FUNCTION_BLOCK FB_System_WP_946
VAR_INPUT
	Freigabe_auto			: BOOL;
	Freigabe_Deakt_auto 	: BOOL;
	Betrieb_Anford_auto		: BOOL;
END_VAR
VAR_OUTPUT
	{attribute 'OPC.UA.DA' := '1'}Steuerung				: ST_System_WP_Steuerung;	
	{attribute 'OPC.UA.DA' := '1'}Stellwert				: ST_System_WP_Stellwert;	
	{attribute 'OPC.UA.DA' := '1'}Zustand					: ST_System_WP_Zustand;	
	{attribute 'OPC.UA.DA' := '1'}Parameter				: ST_System_WP_Parameter;	
END_VAR
VAR
	Waermepumpe_946			: FB_WP;
	Zustandscheck			: FB_System_WP_Zustandscheck;
	Logik					: FB_System_WP_Logik;
	Ablaufsteuerung			: FB_System_WP_Ablaufsteuerung;

	SV_146: FB_SV;
	SV_246: FB_SV;
END_VAR
VAR // added by the converter: edge detectors and wires of the graphical bodies
    _w1, _w2, _w3, _w4 : ANY;
END_VAR

// note: this text did not pass the execution check against the stored diagram
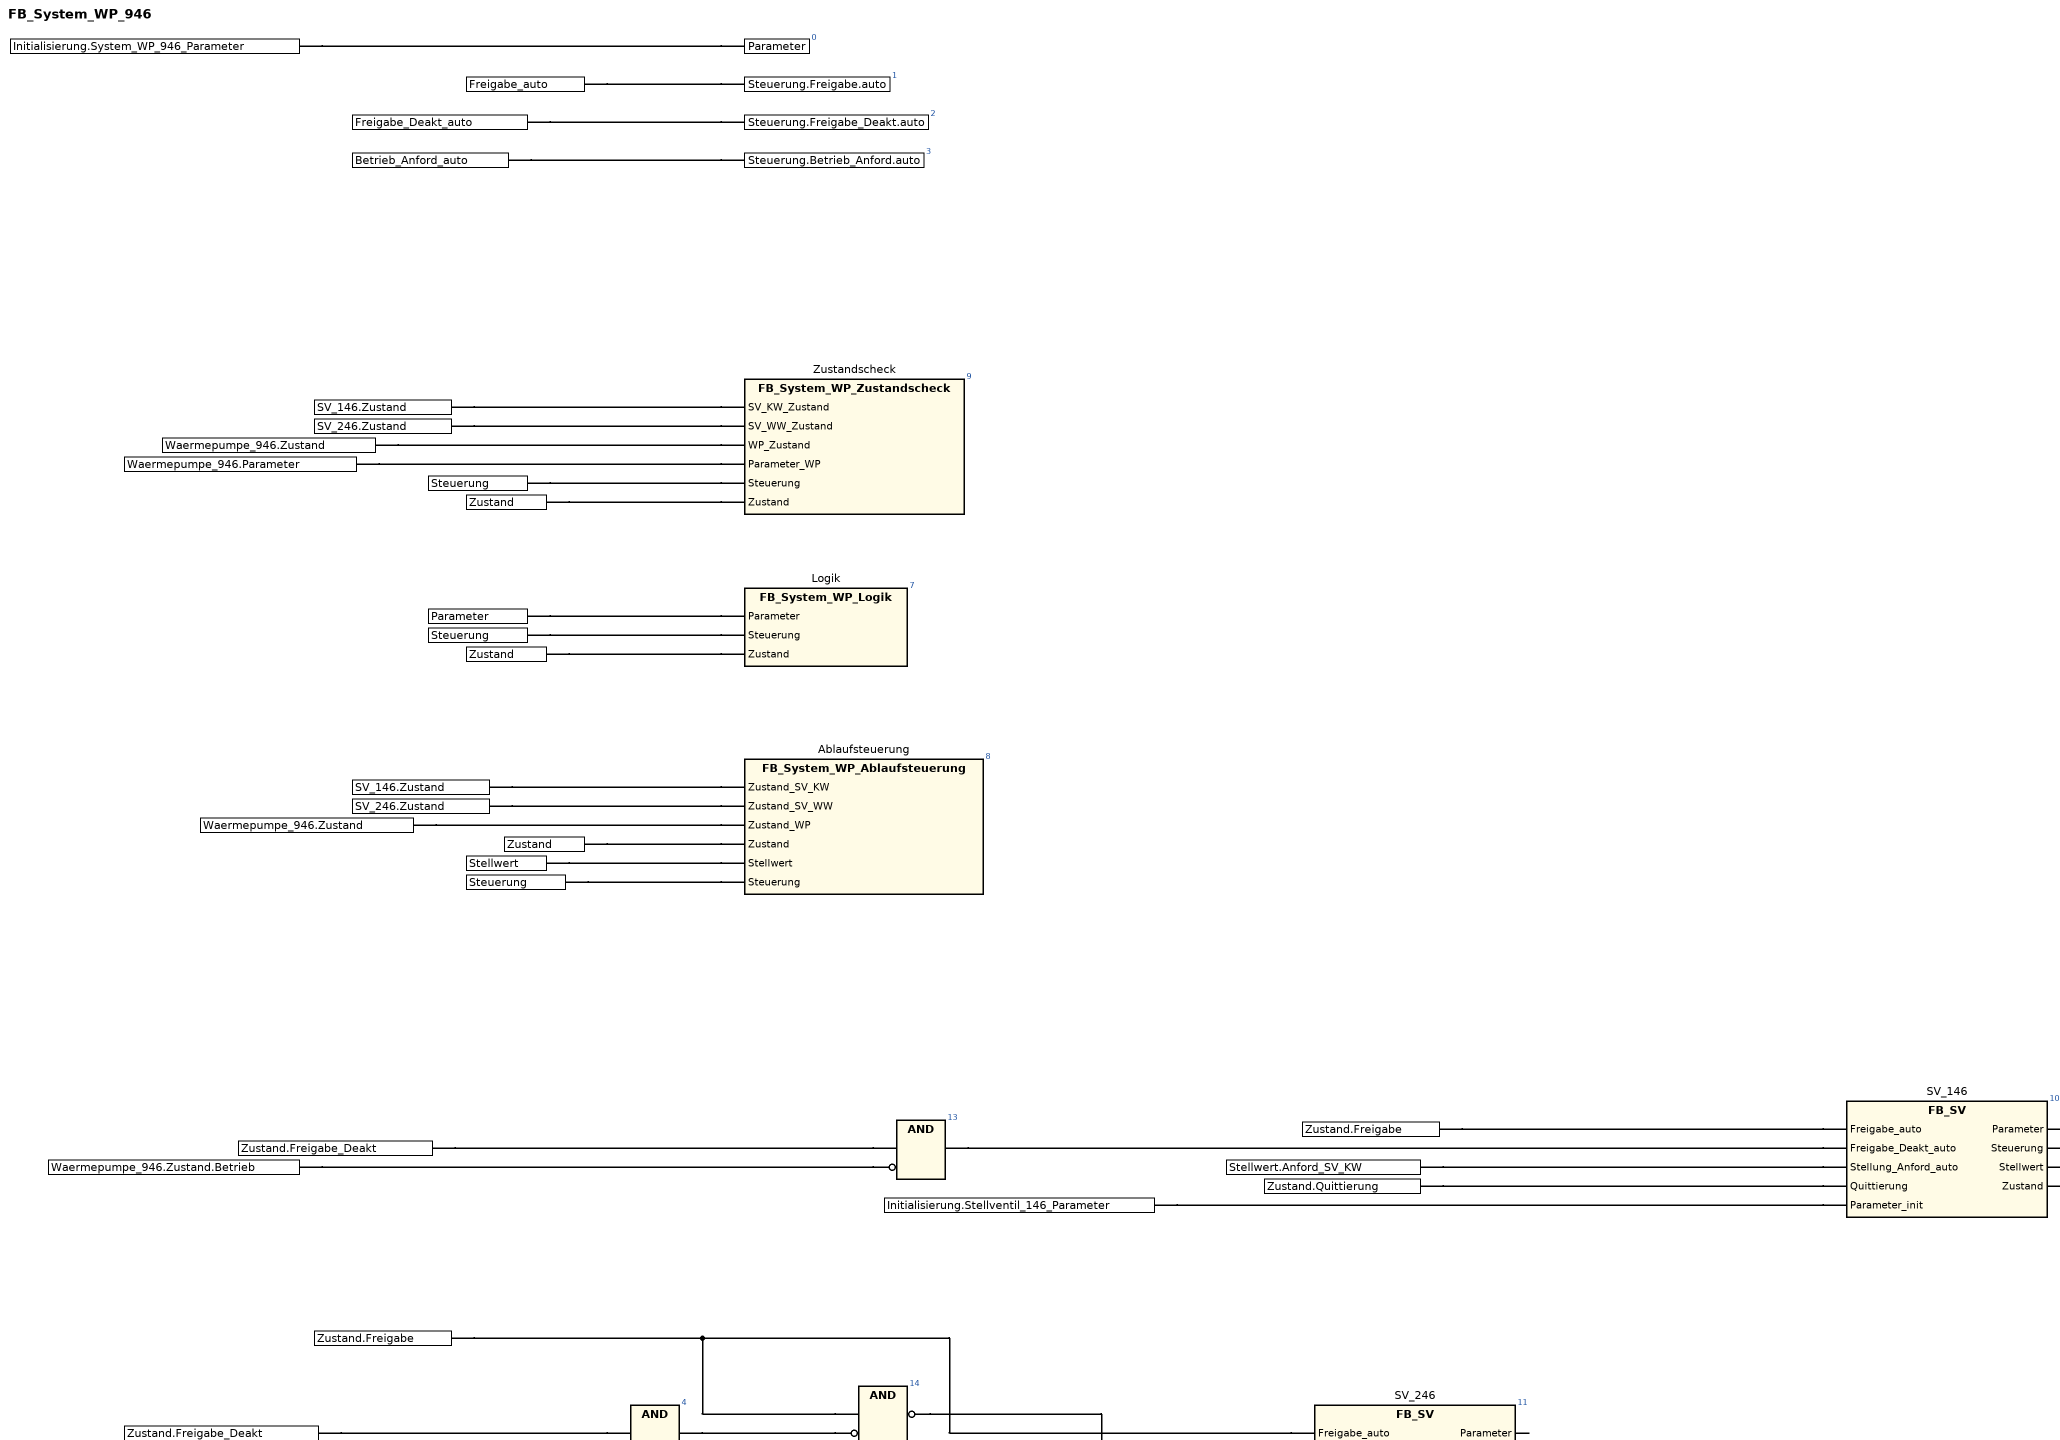
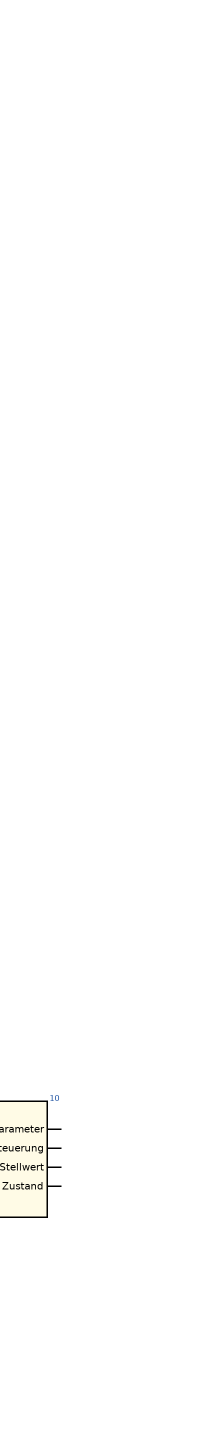
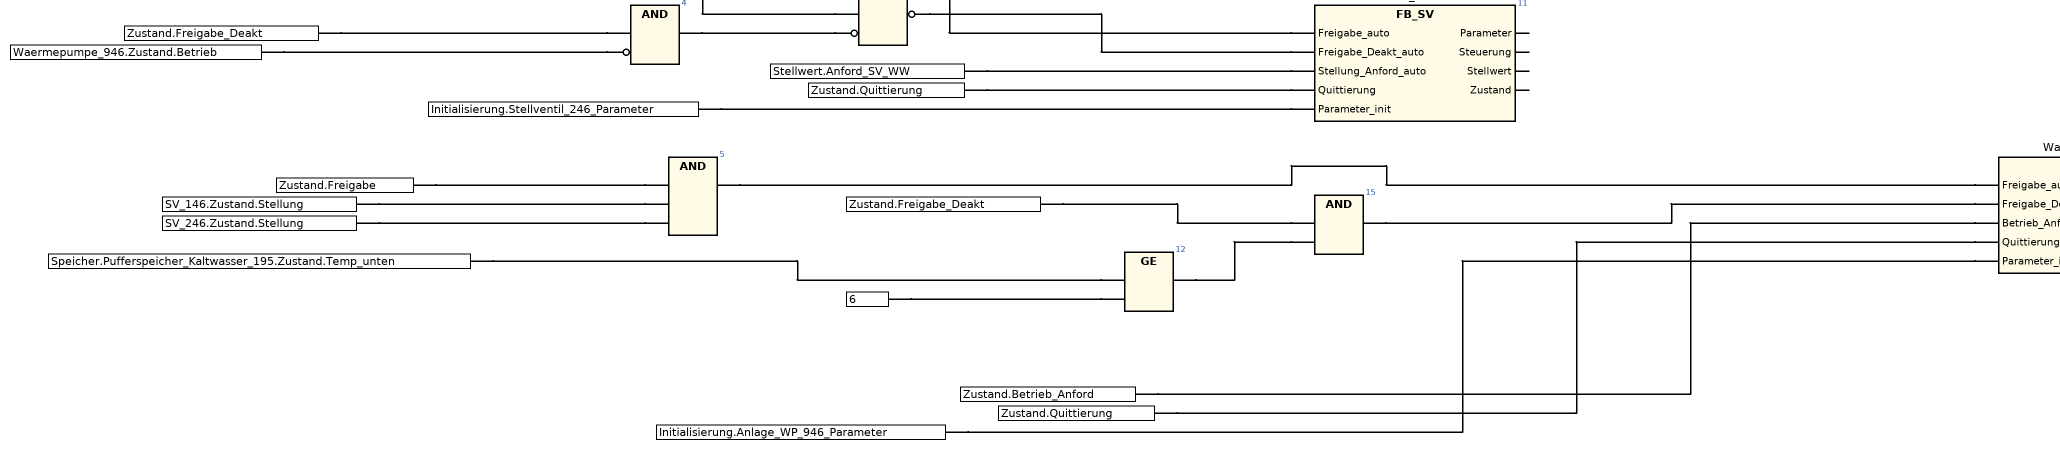
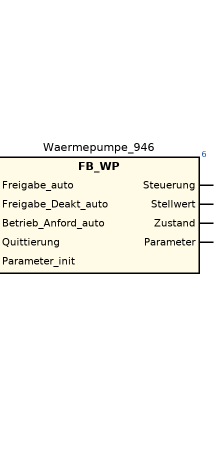
Parameter := Initialisierung.System_WP_946_Parameter;
Steuerung.Freigabe.auto := Freigabe_auto;
Steuerung.Freigabe_Deakt.auto := Freigabe_Deakt_auto;
Steuerung.Betrieb_Anford.auto := Betrieb_Anford_auto;
_w1 := Zustand.Freigabe_Deakt AND NOT Waermepumpe_946.Zustand.Betrieb;
Waermepumpe_946(
    Freigabe_auto := Zustand.Freigabe AND SV_146.Zustand.Stellung AND SV_246.Zustand.Stellung,
    Freigabe_Deakt_auto := _w2,
    Betrieb_Anford_auto := Zustand.Betrieb_Anford,
    Quittierung := Zustand.Quittierung,
    Parameter_init := Initialisierung.Anlage_WP_946_Parameter); // FB_WP
Logik(Parameter := Parameter, Steuerung := Steuerung, Zustand := Zustand); // FB_System_WP_Logik
Ablaufsteuerung(
    Zustand_SV_KW := SV_146.Zustand,
    Zustand_SV_WW := SV_246.Zustand,
    Zustand_WP := Waermepumpe_946.Zustand,
    Zustand := Zustand,
    Stellwert := Stellwert,
    Steuerung := Steuerung); // FB_System_WP_Ablaufsteuerung
Zustandscheck(
    SV_KW_Zustand := SV_146.Zustand,
    SV_WW_Zustand := SV_246.Zustand,
    WP_Zustand := Waermepumpe_946.Zustand,
    Parameter_WP := Waermepumpe_946.Parameter,
    Steuerung := Steuerung,
    Zustand := Zustand); // FB_System_WP_Zustandscheck
SV_146(
    Freigabe_auto := Zustand.Freigabe,
    Freigabe_Deakt_auto := _w3,
    Stellung_Anford_auto := Stellwert.Anford_SV_KW,
    Quittierung := Zustand.Quittierung,
    Parameter_init := Initialisierung.Stellventil_146_Parameter); // FB_SV
SV_246(
    Freigabe_auto := Zustand.Freigabe,
    Freigabe_Deakt_auto := NOT _w4,
    Stellung_Anford_auto := Stellwert.Anford_SV_WW,
    Quittierung := Zustand.Quittierung,
    Parameter_init := Initialisierung.Stellventil_246_Parameter); // FB_SV
_w3 := Zustand.Freigabe_Deakt AND NOT Waermepumpe_946.Zustand.Betrieb;
_w4 := Zustand.Freigabe AND NOT _w1;
_w2 := Zustand.Freigabe_Deakt AND Speicher.Pufferspeicher_Kaltwasser_195.Zustand.Temp_unten >= 6;

END_FUNCTION_BLOCK

(* stored: Version 1.1.0.1, ProductVersion 3.1.4024.9
   POU FB_System_WP_946: Id {9a7c53b7-2d88-433b-bbcd-a2cc30ff8343}, SpecialFunc None *)
